// TIA Portal V19 export
FUNCTION_BLOCK "Valve_Type"   // FB8, LAD
{ S7_Optimized_Access := 'TRUE' }
// stored: MemoryReserve 100, SetENOAutomatically false
   VAR_INPUT
      Auto_OPN : Bool;
      ManOpen : Bool;
      FeedbackFitted : Bool;
      FeedbackTime : Time;
      Close_Feedback : Bool;
      Open_Feedback : Bool;
      Global_Reset : Bool;
      Simulation : Bool;
   END_VAR
   VAR_OUTPUT
      "Valve Open" : Bool;
      "HMI Valve Open" : Bool;
      "HMI Valve Close" : Bool;
      "Valve Open Fault" : Bool;
      "Valve Close Fault" : Bool;
   END_VAR
   VAR_IN_OUT
      "Valve Angle" : Real;
   END_VAR
   VAR
      IEC_Timer_0_Instance { S7_SetPoint := 'True'} : TON_TIME;
      IEC_Timer_0_Instance_1 { S7_SetPoint := 'True'} : TON_TIME;
      "trig 1" : Bool;
      "trig 2" : Bool;
   END_VAR
   VAR_TEMP
      fault_check : Bool;
   END_VAR
   VAR_TEMP   // added for the SCL form of the ladder/FBD networks
      _w1 : Bool;
      _w2 : Bool;
      _w3 : Bool;
      _w4 : Bool;
   END_VAR
BEGIN

REGION Network 1
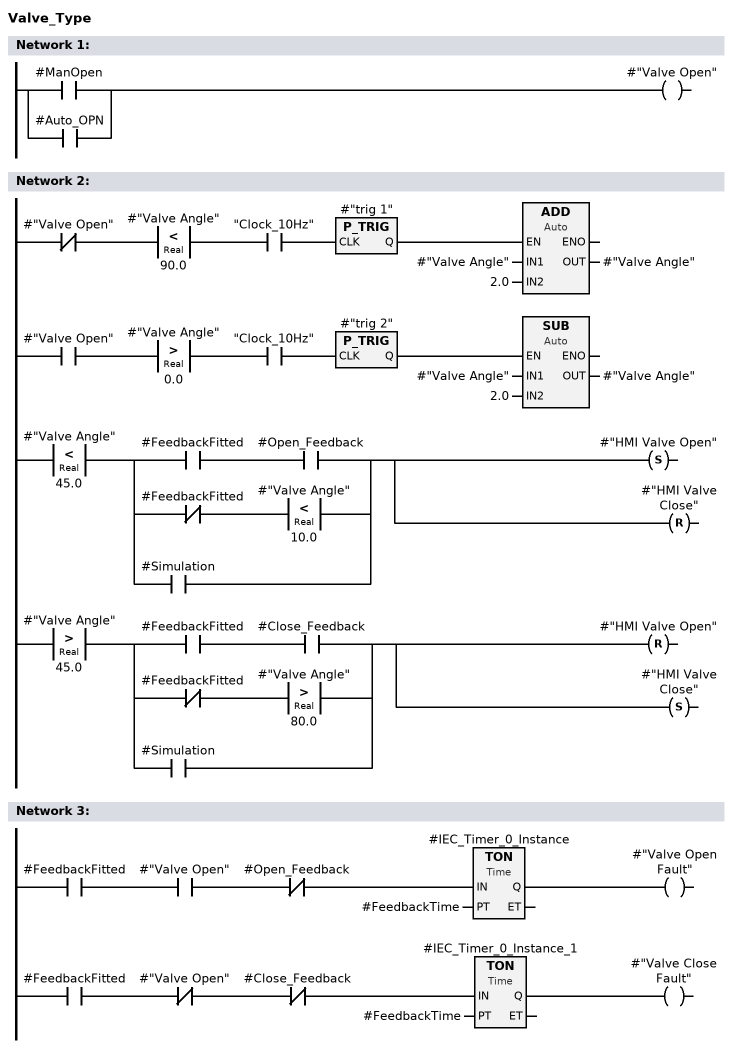
   RUNG wire#powerrail
      Contact( #ManOpen )
      wire#w1
      Coil( #"Valve Open" )
   END_RUNG
   RUNG wire#powerrail
      Contact( #Auto_OPN )
   END_RUNG wire#w1
   // the same network as SCL:
   #"Valve Open" := #ManOpen OR #Auto_OPN;
END_REGION

REGION Network 2
   RUNG wire#powerrail
      I_Contact( #"Valve Open" )
      { S7_Templates := "SrcType := Real" } LT_Contact(in1 := #"Valve Angle", in2 := 90.0)
      Contact( "Clock_10Hz" )
      P_Trig( #"trig 1" )
      Add(in1 := #"Valve Angle", in2 := 2.0, out => #"Valve Angle")
   END_RUNG
   RUNG wire#powerrail
      Contact( #"Valve Open" )
      { S7_Templates := "SrcType := Real" } GT_Contact(in1 := #"Valve Angle", in2 := 0.0)
      Contact( "Clock_10Hz" )
      P_Trig( #"trig 2" )
      Sub(in1 := #"Valve Angle", in2 := 2.0, out => #"Valve Angle")
   END_RUNG
   RUNG wire#powerrail
      { S7_Templates := "SrcType := Real" } LT_Contact(in1 := #"Valve Angle", in2 := 45.0)
      wire#w1
      Contact( #FeedbackFitted )
      Contact( #Open_Feedback )
      wire#w2
      S_Coil( #"HMI Valve Open" )
   END_RUNG
   RUNG wire#w1
      I_Contact( #FeedbackFitted )
      { S7_Templates := "SrcType := Real" } LT_Contact(in1 := #"Valve Angle", in2 := 10.0)
   END_RUNG wire#w2
   RUNG wire#w1
      Contact( #Simulation )
   END_RUNG wire#w2
   RUNG wire#w2
      R_Coil( #"HMI Valve Close" )
   END_RUNG
   RUNG wire#powerrail
      { S7_Templates := "SrcType := Real" } GT_Contact(in1 := #"Valve Angle", in2 := 45.0)
      wire#w3
      Contact( #FeedbackFitted )
      Contact( #Close_Feedback )
      wire#w4
      R_Coil( #"HMI Valve Open" )
   END_RUNG
   RUNG wire#w3
      I_Contact( #FeedbackFitted )
      { S7_Templates := "SrcType := Real" } GT_Contact(in1 := #"Valve Angle", in2 := 80.0)
   END_RUNG wire#w4
   RUNG wire#w3
      Contact( #Simulation )
   END_RUNG wire#w4
   RUNG wire#w4
      S_Coil( #"HMI Valve Close" )
   END_RUNG
   // the same network as SCL:
   #_w1 := NOT #"Valve Open" AND (#"Valve Angle" < 90.0) AND "Clock_10Hz";
   #_w2 := #_w1 AND NOT #"trig 1";   // rising edge
   #"trig 1" := #_w1;
   IF #_w2 THEN #"Valve Angle" := #"Valve Angle" + 2.0; END_IF;
   #_w3 := #"Valve Open" AND (#"Valve Angle" > 0.0) AND "Clock_10Hz";
   #_w4 := #_w3 AND NOT #"trig 2";   // rising edge
   #"trig 2" := #_w3;
   IF #_w4 THEN #"Valve Angle" := #"Valve Angle" - 2.0; END_IF;
   IF (#"Valve Angle" < 45.0) AND ((#FeedbackFitted AND #Open_Feedback) OR (NOT #FeedbackFitted AND (#"Valve Angle" < 10.0)) OR #Simulation) THEN
       #"HMI Valve Open" := TRUE;
       #"HMI Valve Close" := FALSE;
   END_IF;
   IF (#"Valve Angle" > 45.0) AND ((#FeedbackFitted AND #Close_Feedback) OR (NOT #FeedbackFitted AND (#"Valve Angle" > 80.0)) OR #Simulation) THEN
       #"HMI Valve Open" := FALSE;
       #"HMI Valve Close" := TRUE;
   END_IF;
END_REGION

REGION Network 3
   RUNG wire#powerrail
      Contact( #FeedbackFitted )
      Contact( #"Valve Open" )
      I_Contact( #Open_Feedback )
      { S7_Templates := "time_type := Time" } #IEC_Timer_0_Instance.TON(pt := #FeedbackTime, et =>)
      Coil( #"Valve Open Fault" )
   END_RUNG
   RUNG wire#powerrail
      Contact( #FeedbackFitted )
      I_Contact( #"Valve Open" )
      I_Contact( #Close_Feedback )
      { S7_Templates := "time_type := Time" } #IEC_Timer_0_Instance_1.TON(pt := #FeedbackTime, et =>)
      Coil( #"Valve Close Fault" )
   END_RUNG
   // the same network as SCL:
   #IEC_Timer_0_Instance(IN := #FeedbackFitted AND #"Valve Open" AND NOT #Open_Feedback, PT := #FeedbackTime);   // TON
   #"Valve Open Fault" := #IEC_Timer_0_Instance.Q;
   #IEC_Timer_0_Instance_1(IN := #FeedbackFitted AND NOT #"Valve Open" AND NOT #Close_Feedback,   // TON
                           PT := #FeedbackTime);
   #"Valve Close Fault" := #IEC_Timer_0_Instance_1.Q;
END_REGION
END_FUNCTION_BLOCK
